// TIA Portal V20 export
FUNCTION_BLOCK "LER_StackMainCommand"   // FB95, LAD
// stored: Access Published, MemoryReserve 100, SetENOAutomatically false
   VAR_INPUT
      enable : Bool;
      reset : Bool;
      rollerCathodePos : Bool;
      rollerAnodePos : Bool;
      timeOffSet { ExternalAccessible := 'False'; ExternalVisible := 'False'; ExternalWritable := 'False'} : Time;
      motionStatus : Struct
         StopRequest : Bool := FALSE;
         Busy : Struct
            TotalBusy : Bool;
            CalculateBusy : Bool;
            SemiStepBusy : Bool;
            FullStepBusy : Bool;
            AutoBusy : Bool;
            CycleStopBusy : Bool;
            FastStopBusy : Bool;
            ResetBusy : Bool;
         END_STRUCT;
         Done : Struct
            TotalDone : Bool;
            CalculateDone : Bool;
            SemiStepDone : Bool;
            FullStepDone : Bool;
            AutoDone : Bool;
            CycleStopDone : Bool;
            FastStopDone : Bool;
            ResetDone : Bool;
         END_STRUCT;
         Error : Bool := FALSE;
         ErrorID : DWord := 16#0000_0000;
         NowCmd : DInt := 0;
         BeforeCmd : DInt := 0;
         NowStep : DInt := 160;
         BeforeStep : DInt := 180;
      END_STRUCT;
      unitStatus : "LAF_typeUnitStatus";
   END_VAR
   VAR_OUTPUT
      direction : Bool;
      motionCommands : Struct
         Calculate : Bool := FALSE;
         SemiStep : Bool := FALSE;
         FullStep : Bool := FALSE;
         Auto : Bool := FALSE;
         SepaClean : Bool;
         CycleStop : Bool := FALSE;
         FastStop : Bool;
         Reset : Bool := FALSE;
      END_STRUCT;
   END_VAR
   VAR_IN_OUT
      motionInterface : Struct
         Calculate : Bool;
         SemiStep : Bool;
         FullStep : Bool;
         AutoReady : Bool;
         AutoStart : Bool;
         StopMotion : Bool;
         StopForCalculate : Bool;
         Reset : Bool;
      END_STRUCT;
   END_VAR
   VAR
      statTonTime { ExternalAccessible := 'False'; ExternalVisible := 'False'; ExternalWritable := 'False'} : Array[0..999] of TON_TIME;
      statPulse { ExternalAccessible := 'False'; ExternalVisible := 'False'; ExternalWritable := 'False'} : Array[0..999] of Bool;
      statAction { ExternalAccessible := 'False'; ExternalVisible := 'False'; ExternalWritable := 'False'} : Array[0..999] of Bool;
      statStep { ExternalAccessible := 'False'; ExternalVisible := 'False'; ExternalWritable := 'False'} : DInt;
      statMotionStatus { ExternalAccessible := 'False'; ExternalVisible := 'False'; ExternalWritable := 'False'} : DInt;
   END_VAR
   VAR CONSTANT
      delayTime : Time := T#0ms;
   END_VAR
   VAR_TEMP   // added for the SCL form of the ladder/FBD networks
      _w1 : Bool;
      _w2 : Bool;
      _w3 : Bool;
      _w4 : Bool;
      _w5 : Bool;
      _w6 : Bool;
   END_VAR
BEGIN

REGION Network 1: ******************** Motion Operation ********************
END_REGION

REGION Network 2: STEP[0] : Motion Operation Condition
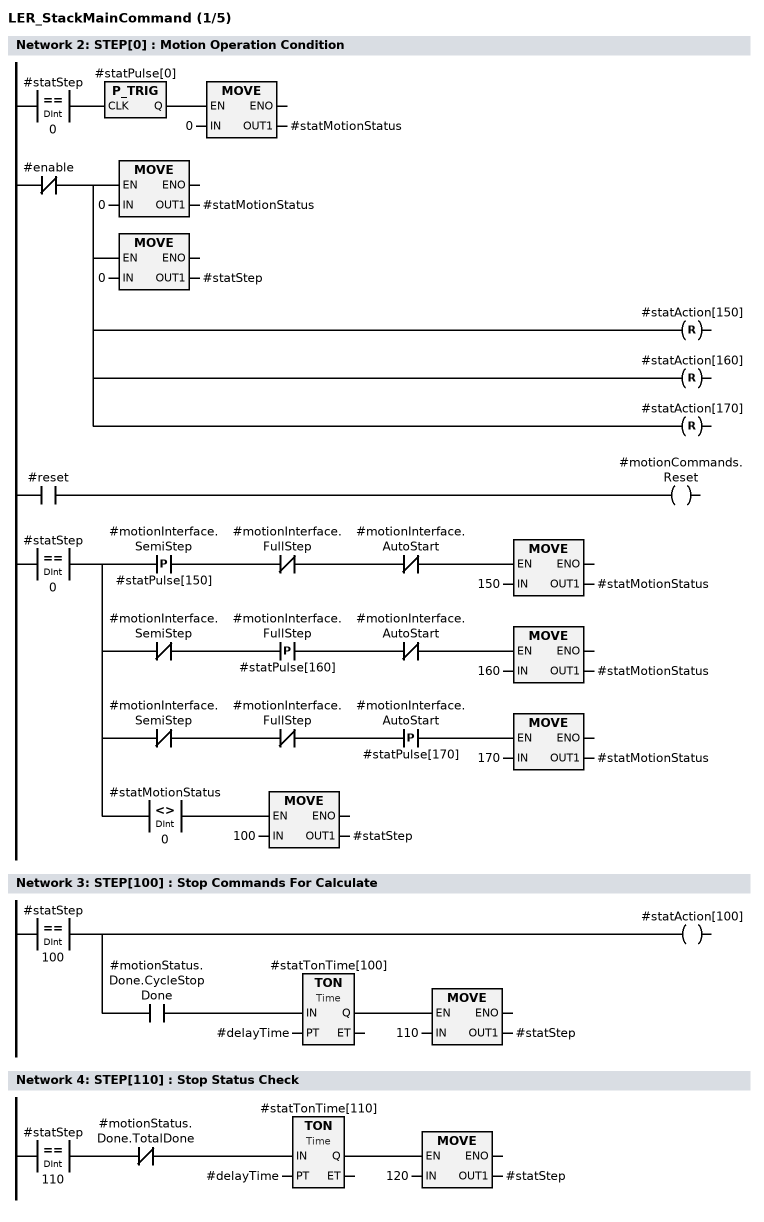
   RUNG wire#powerrail
      { S7_Templates := "SrcType := DInt" } EQ_Contact(in1 := #statStep, in2 := 0)
      P_Trig( #statPulse[0] )
      Move(in := 0, out1 => #statMotionStatus)
   END_RUNG
   RUNG wire#powerrail
      I_Contact( #enable )
      wire#w1
      Move(in := 0, out1 => #statMotionStatus)
   END_RUNG
   RUNG wire#w1
      Move(in := 0, out1 => #statStep)
   END_RUNG
   RUNG wire#w1
      R_Coil( #statAction[150] )
   END_RUNG
   RUNG wire#w1
      R_Coil( #statAction[160] )
   END_RUNG
   RUNG wire#w1
      R_Coil( #statAction[170] )
   END_RUNG
   RUNG wire#powerrail
      Contact( #reset )
      Coil( #motionCommands.Reset )
   END_RUNG
   RUNG wire#powerrail
      { S7_Templates := "SrcType := DInt" } EQ_Contact(in1 := #statStep, in2 := 0)
      wire#w2
      P_Contact(operand := #motionInterface.SemiStep, bit := #statPulse[150])
      I_Contact( #motionInterface.FullStep )
      I_Contact( #motionInterface.AutoStart )
      Move(in := 150, out1 => #statMotionStatus)
   END_RUNG
   RUNG wire#w2
      I_Contact( #motionInterface.SemiStep )
      P_Contact(operand := #motionInterface.FullStep, bit := #statPulse[160])
      I_Contact( #motionInterface.AutoStart )
      Move(in := 160, out1 => #statMotionStatus)
   END_RUNG
   RUNG wire#w2
      I_Contact( #motionInterface.SemiStep )
      I_Contact( #motionInterface.FullStep )
      P_Contact(operand := #motionInterface.AutoStart, bit := #statPulse[170])
      Move(in := 170, out1 => #statMotionStatus)
   END_RUNG
   RUNG wire#w2
      { S7_Templates := "SrcType := DInt" } NE_Contact(in1 := #statMotionStatus, in2 := 0)
      Move(in := 100, out1 => #statStep)
   END_RUNG
   // the same network as SCL:
   #_w1 := #statStep = 0;
   #_w2 := #_w1 AND NOT #statPulse[0];   // rising edge
   #statPulse[0] := #_w1;
   IF #_w2 THEN #statMotionStatus := 0; END_IF;
   IF NOT #enable THEN
       #statMotionStatus := 0;
       #statStep := 0;
       #statAction[150] := FALSE;
       #statAction[160] := FALSE;
       #statAction[170] := FALSE;
   END_IF;
   #motionCommands.Reset := #reset;
   #_w3 := #statStep = 0;
   #_w4 := #_w3 AND #motionInterface.SemiStep AND NOT #statPulse[150];   // rising edge of #motionInterface.SemiStep
   #statPulse[150] := #motionInterface.SemiStep;
   IF #_w4 AND NOT #motionInterface.FullStep AND NOT #motionInterface.AutoStart THEN
       #statMotionStatus := 150;
   END_IF;
   #_w5 := #_w3 AND NOT #motionInterface.SemiStep AND #motionInterface.FullStep AND NOT #statPulse[160];   // rising edge of #motionInterface.FullStep
   #statPulse[160] := #motionInterface.FullStep;
   IF #_w5 AND NOT #motionInterface.AutoStart THEN #statMotionStatus := 160; END_IF;
   #_w6 := #_w3 AND NOT #motionInterface.SemiStep AND NOT #motionInterface.FullStep AND #motionInterface.AutoStart AND NOT #statPulse[170];   // rising edge of #motionInterface.AutoStart
   #statPulse[170] := #motionInterface.AutoStart;
   IF #_w6 THEN #statMotionStatus := 170; END_IF;
   IF #_w3 AND (#statMotionStatus <> 0) THEN #statStep := 100; END_IF;
END_REGION

REGION Network 3: STEP[100] : Stop Commands For Calculate
   RUNG wire#powerrail
      { S7_Templates := "SrcType := DInt" } EQ_Contact(in1 := #statStep, in2 := 100)
      wire#w1
      Coil( #statAction[100] )
   END_RUNG
   RUNG wire#w1
      Contact( #motionStatus.Done.CycleStopDone )
      { S7_Templates := "time_type := Time" } #statTonTime[100].TON(pt := #delayTime, et =>)
      Move(in := 110, out1 => #statStep)
   END_RUNG
   // the same network as SCL:
   #statAction[100] := #statStep = 100;
   #statTonTime[100].TON(IN := (#statStep = 100) AND #motionStatus.Done.CycleStopDone, PT := #delayTime);
   IF #statTonTime[100].Q THEN #statStep := 110; END_IF;
END_REGION

REGION Network 4: STEP[110] : Stop Status Check
   RUNG wire#powerrail
      { S7_Templates := "SrcType := DInt" } EQ_Contact(in1 := #statStep, in2 := 110)
      I_Contact( #motionStatus.Done.TotalDone )
      { S7_Templates := "time_type := Time" } #statTonTime[110].TON(pt := #delayTime, et =>)
      Move(in := 120, out1 => #statStep)
   END_RUNG
   // the same network as SCL:
   #statTonTime[110].TON(IN := (#statStep = 110) AND NOT #motionStatus.Done.TotalDone, PT := #delayTime);
   IF #statTonTime[110].Q THEN #statStep := 120; END_IF;
END_REGION

REGION Network 5: STEP[120] : Parameter Direction Select
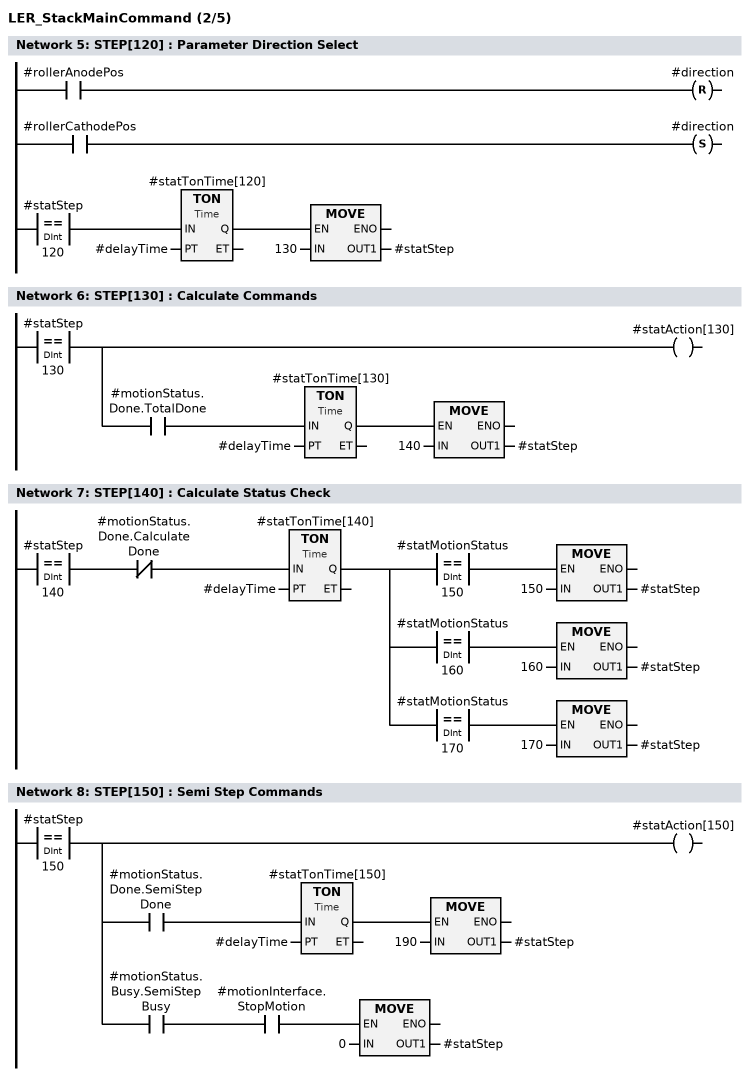
   RUNG wire#powerrail
      Contact( #rollerAnodePos )
      R_Coil( #direction )
   END_RUNG
   RUNG wire#powerrail
      Contact( #rollerCathodePos )
      S_Coil( #direction )
   END_RUNG
   RUNG wire#powerrail
      { S7_Templates := "SrcType := DInt" } EQ_Contact(in1 := #statStep, in2 := 120)
      { S7_Templates := "time_type := Time" } #statTonTime[120].TON(pt := #delayTime, et =>)
      Move(in := 130, out1 => #statStep)
   END_RUNG
   // the same network as SCL:
   IF #rollerAnodePos THEN #direction := FALSE; END_IF;
   IF #rollerCathodePos THEN #direction := TRUE; END_IF;
   #statTonTime[120].TON(IN := #statStep = 120, PT := #delayTime);
   IF #statTonTime[120].Q THEN #statStep := 130; END_IF;
END_REGION

REGION Network 6: STEP[130] : Calculate Commands
   RUNG wire#powerrail
      { S7_Templates := "SrcType := DInt" } EQ_Contact(in1 := #statStep, in2 := 130)
      wire#w1
      Coil( #statAction[130] )
   END_RUNG
   RUNG wire#w1
      Contact( #motionStatus.Done.TotalDone )
      { S7_Templates := "time_type := Time" } #statTonTime[130].TON(pt := #delayTime, et =>)
      Move(in := 140, out1 => #statStep)
   END_RUNG
   // the same network as SCL:
   #statAction[130] := #statStep = 130;
   #statTonTime[130].TON(IN := (#statStep = 130) AND #motionStatus.Done.TotalDone, PT := #delayTime);
   IF #statTonTime[130].Q THEN #statStep := 140; END_IF;
END_REGION

REGION Network 7: STEP[140] : Calculate Status Check
   RUNG wire#powerrail
      { S7_Templates := "SrcType := DInt" } EQ_Contact(in1 := #statStep, in2 := 140)
      I_Contact( #motionStatus.Done.CalculateDone )
      { S7_Templates := "time_type := Time" } #statTonTime[140].TON(pt := #delayTime, et =>)
      wire#w1
      { S7_Templates := "SrcType := DInt" } EQ_Contact(in1 := #statMotionStatus, in2 := 150)
      Move(in := 150, out1 => #statStep)
   END_RUNG
   RUNG wire#w1
      { S7_Templates := "SrcType := DInt" } EQ_Contact(in1 := #statMotionStatus, in2 := 160)
      Move(in := 160, out1 => #statStep)
   END_RUNG
   RUNG wire#w1
      { S7_Templates := "SrcType := DInt" } EQ_Contact(in1 := #statMotionStatus, in2 := 170)
      Move(in := 170, out1 => #statStep)
   END_RUNG
   // the same network as SCL:
   #statTonTime[140].TON(IN := (#statStep = 140) AND NOT #motionStatus.Done.CalculateDone, PT := #delayTime);
   IF #statTonTime[140].Q AND (#statMotionStatus = 150) THEN #statStep := 150; END_IF;
   IF #statTonTime[140].Q AND (#statMotionStatus = 160) THEN #statStep := 160; END_IF;
   IF #statTonTime[140].Q AND (#statMotionStatus = 170) THEN #statStep := 170; END_IF;
END_REGION

REGION Network 8: STEP[150] : Semi Step Commands
   RUNG wire#powerrail
      { S7_Templates := "SrcType := DInt" } EQ_Contact(in1 := #statStep, in2 := 150)
      wire#w1
      Coil( #statAction[150] )
   END_RUNG
   RUNG wire#w1
      Contact( #motionStatus.Done.SemiStepDone )
      { S7_Templates := "time_type := Time" } #statTonTime[150].TON(pt := #delayTime, et =>)
      Move(in := 190, out1 => #statStep)
   END_RUNG
   RUNG wire#w1
      Contact( #motionStatus.Busy.SemiStepBusy )
      Contact( #motionInterface.StopMotion )
      Move(in := 0, out1 => #statStep)
   END_RUNG
   // the same network as SCL:
   #statAction[150] := #statStep = 150;
   #statTonTime[150].TON(IN := (#statStep = 150) AND #motionStatus.Done.SemiStepDone, PT := #delayTime);
   #_w1 := #statStep = 150;
   IF #statTonTime[150].Q THEN #statStep := 190; END_IF;
   IF #_w1 AND #motionStatus.Busy.SemiStepBusy AND #motionInterface.StopMotion THEN #statStep := 0; END_IF;
END_REGION

REGION Network 9: STEP[160] : Full Step Commands
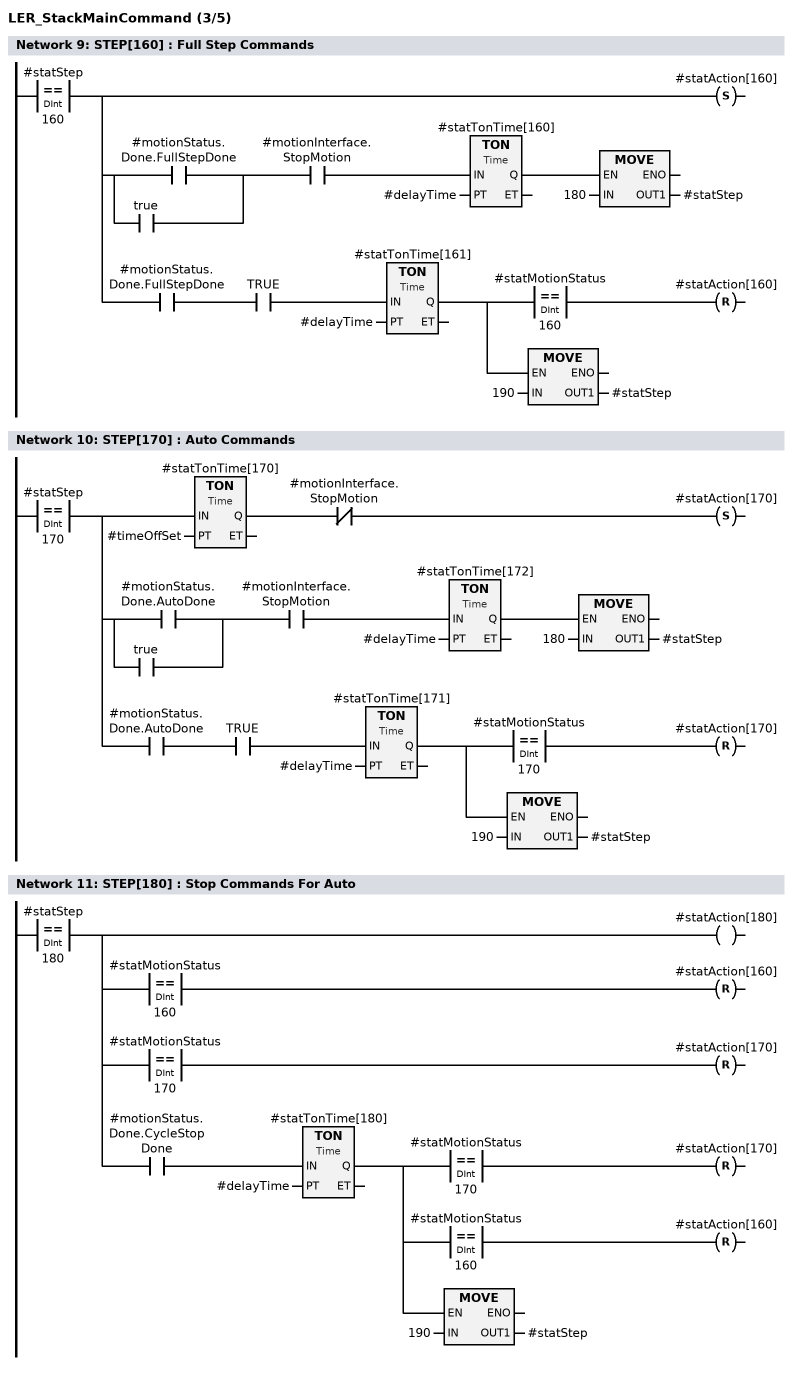
   RUNG wire#powerrail
      { S7_Templates := "SrcType := DInt" } EQ_Contact(in1 := #statStep, in2 := 160)
      wire#w1
      S_Coil( #statAction[160] )
   END_RUNG
   RUNG wire#w1
      Contact( #motionStatus.Done.FullStepDone )
      wire#w2
      Contact( #motionInterface.StopMotion )
      { S7_Templates := "time_type := Time" } #statTonTime[160].TON(pt := #delayTime, et =>)
      Move(in := 180, out1 => #statStep)
   END_RUNG
   RUNG wire#w1
      Contact( true )
   END_RUNG wire#w2
   RUNG wire#w1
      Contact( #motionStatus.Done.FullStepDone )
      Contact( TRUE )
      { S7_Templates := "time_type := Time" } #statTonTime[161].TON(pt := #delayTime, et =>)
      wire#w3
      { S7_Templates := "SrcType := DInt" } EQ_Contact(in1 := #statMotionStatus, in2 := 160)
      R_Coil( #statAction[160] )
   END_RUNG
   RUNG wire#w3
      Move(in := 190, out1 => #statStep)
   END_RUNG
   // the same network as SCL:
   #_w1 := #statStep = 160;
   IF #_w1 THEN #statAction[160] := TRUE; END_IF;
   #statTonTime[160].TON(IN := #_w1 AND (#motionStatus.Done.FullStepDone OR true) AND #motionInterface.StopMotion,
                         PT := #delayTime);
   IF #statTonTime[160].Q THEN #statStep := 180; END_IF;
   #statTonTime[161].TON(IN := #_w1 AND #motionStatus.Done.FullStepDone AND TRUE, PT := #delayTime);
   IF #statTonTime[161].Q AND (#statMotionStatus = 160) THEN #statAction[160] := FALSE; END_IF;
   IF #statTonTime[161].Q THEN #statStep := 190; END_IF;
END_REGION

REGION Network 10: STEP[170] : Auto Commands
   RUNG wire#powerrail
      { S7_Templates := "SrcType := DInt" } EQ_Contact(in1 := #statStep, in2 := 170)
      wire#w1
      { S7_Templates := "time_type := Time" } #statTonTime[170].TON(pt := #timeOffSet, et =>)
      I_Contact( #motionInterface.StopMotion )
      S_Coil( #statAction[170] )
   END_RUNG
   RUNG wire#w1
      Contact( #motionStatus.Done.AutoDone )
      wire#w2
      Contact( #motionInterface.StopMotion )
      { S7_Templates := "time_type := Time" } #statTonTime[172].TON(pt := #delayTime, et =>)
      Move(in := 180, out1 => #statStep)
   END_RUNG
   RUNG wire#w1
      Contact( true )
   END_RUNG wire#w2
   RUNG wire#w1
      Contact( #motionStatus.Done.AutoDone )
      Contact( TRUE )
      { S7_Templates := "time_type := Time" } #statTonTime[171].TON(pt := #delayTime, et =>)
      wire#w3
      { S7_Templates := "SrcType := DInt" } EQ_Contact(in1 := #statMotionStatus, in2 := 170)
      R_Coil( #statAction[170] )
   END_RUNG
   RUNG wire#w3
      Move(in := 190, out1 => #statStep)
   END_RUNG
   // the same network as SCL:
   #_w1 := #statStep = 170;
   #statTonTime[170].TON(IN := #_w1, PT := #timeOffSet);
   IF #statTonTime[170].Q AND NOT #motionInterface.StopMotion THEN #statAction[170] := TRUE; END_IF;
   #statTonTime[172].TON(IN := #_w1 AND (#motionStatus.Done.AutoDone OR true) AND #motionInterface.StopMotion,
                         PT := #delayTime);
   IF #statTonTime[172].Q THEN #statStep := 180; END_IF;
   #statTonTime[171].TON(IN := #_w1 AND #motionStatus.Done.AutoDone AND TRUE, PT := #delayTime);
   IF #statTonTime[171].Q AND (#statMotionStatus = 170) THEN #statAction[170] := FALSE; END_IF;
   IF #statTonTime[171].Q THEN #statStep := 190; END_IF;
END_REGION

REGION Network 11: STEP[180] : Stop Commands For Auto
   RUNG wire#powerrail
      { S7_Templates := "SrcType := DInt" } EQ_Contact(in1 := #statStep, in2 := 180)
      wire#w1
      Coil( #statAction[180] )
   END_RUNG
   RUNG wire#w1
      { S7_Templates := "SrcType := DInt" } EQ_Contact(in1 := #statMotionStatus, in2 := 160)
      R_Coil( #statAction[160] )
   END_RUNG
   RUNG wire#w1
      { S7_Templates := "SrcType := DInt" } EQ_Contact(in1 := #statMotionStatus, in2 := 170)
      R_Coil( #statAction[170] )
   END_RUNG
   RUNG wire#w1
      Contact( #motionStatus.Done.CycleStopDone )
      { S7_Templates := "time_type := Time" } #statTonTime[180].TON(pt := #delayTime, et =>)
      wire#w2
      { S7_Templates := "SrcType := DInt" } EQ_Contact(in1 := #statMotionStatus, in2 := 170)
      R_Coil( #statAction[170] )
   END_RUNG
   RUNG wire#w2
      { S7_Templates := "SrcType := DInt" } EQ_Contact(in1 := #statMotionStatus, in2 := 160)
      R_Coil( #statAction[160] )
   END_RUNG
   RUNG wire#w2
      Move(in := 190, out1 => #statStep)
   END_RUNG
   // the same network as SCL:
   #statAction[180] := #statStep = 180;
   IF (#statStep = 180) AND (#statMotionStatus = 160) THEN #statAction[160] := FALSE; END_IF;
   IF (#statStep = 180) AND (#statMotionStatus = 170) THEN #statAction[170] := FALSE; END_IF;
   #statTonTime[180].TON(IN := (#statStep = 180) AND #motionStatus.Done.CycleStopDone, PT := #delayTime);
   IF #statTonTime[180].Q AND (#statMotionStatus = 170) THEN #statAction[170] := FALSE; END_IF;
   IF #statTonTime[180].Q AND (#statMotionStatus = 160) THEN #statAction[160] := FALSE; END_IF;
   IF #statTonTime[180].Q THEN #statStep := 190; END_IF;
END_REGION

REGION Network 12: STEP[190] : Motion Operation Complete
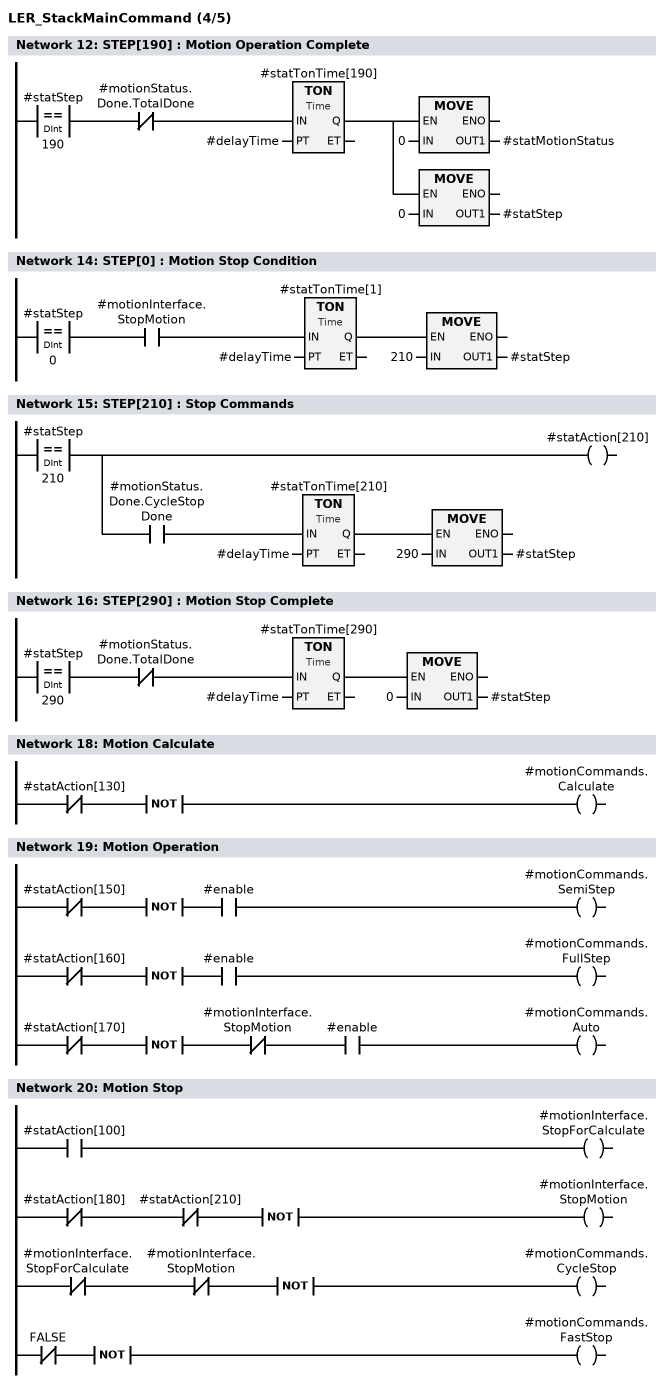
   RUNG wire#powerrail
      { S7_Templates := "SrcType := DInt" } EQ_Contact(in1 := #statStep, in2 := 190)
      I_Contact( #motionStatus.Done.TotalDone )
      { S7_Templates := "time_type := Time" } #statTonTime[190].TON(pt := #delayTime, et =>)
      wire#w1
      Move(in := 0, out1 => #statMotionStatus)
   END_RUNG
   RUNG wire#w1
      Move(in := 0, out1 => #statStep)
   END_RUNG
   // the same network as SCL:
   #statTonTime[190].TON(IN := (#statStep = 190) AND NOT #motionStatus.Done.TotalDone, PT := #delayTime);
   IF #statTonTime[190].Q THEN
       #statMotionStatus := 0;
       #statStep := 0;
   END_IF;
END_REGION

REGION Network 13: ******************** Motion Stop ********************
END_REGION

REGION Network 14: STEP[0] : Motion Stop Condition
   RUNG wire#powerrail
      { S7_Templates := "SrcType := DInt" } EQ_Contact(in1 := #statStep, in2 := 0)
      Contact( #motionInterface.StopMotion )
      { S7_Templates := "time_type := Time" } #statTonTime[1].TON(pt := #delayTime, et =>)
      Move(in := 210, out1 => #statStep)
   END_RUNG
   // the same network as SCL:
   #statTonTime[1].TON(IN := (#statStep = 0) AND #motionInterface.StopMotion, PT := #delayTime);
   IF #statTonTime[1].Q THEN #statStep := 210; END_IF;
END_REGION

REGION Network 15: STEP[210] : Stop Commands
   RUNG wire#powerrail
      { S7_Templates := "SrcType := DInt" } EQ_Contact(in1 := #statStep, in2 := 210)
      wire#w1
      Coil( #statAction[210] )
   END_RUNG
   RUNG wire#w1
      Contact( #motionStatus.Done.CycleStopDone )
      { S7_Templates := "time_type := Time" } #statTonTime[210].TON(pt := #delayTime, et =>)
      Move(in := 290, out1 => #statStep)
   END_RUNG
   // the same network as SCL:
   #statAction[210] := #statStep = 210;
   #statTonTime[210].TON(IN := (#statStep = 210) AND #motionStatus.Done.CycleStopDone, PT := #delayTime);
   IF #statTonTime[210].Q THEN #statStep := 290; END_IF;
END_REGION

REGION Network 16: STEP[290] : Motion Stop Complete
   RUNG wire#powerrail
      { S7_Templates := "SrcType := DInt" } EQ_Contact(in1 := #statStep, in2 := 290)
      I_Contact( #motionStatus.Done.TotalDone )
      { S7_Templates := "time_type := Time" } #statTonTime[290].TON(pt := #delayTime, et =>)
      Move(in := 0, out1 => #statStep)
   END_RUNG
   // the same network as SCL:
   #statTonTime[290].TON(IN := (#statStep = 290) AND NOT #motionStatus.Done.TotalDone, PT := #delayTime);
   IF #statTonTime[290].Q THEN #statStep := 0; END_IF;
END_REGION

REGION Network 17: ******************** Motion Commands ********************
END_REGION

REGION Network 18: Motion Calculate
   RUNG wire#powerrail
      I_Contact( #statAction[130] )
      Not()
      Coil( #motionCommands.Calculate )
   END_RUNG
   // the same network as SCL:
   #motionCommands.Calculate := NOT (NOT #statAction[130]);
END_REGION

REGION Network 19: Motion Operation
   RUNG wire#powerrail
      I_Contact( #statAction[150] )
      Not()
      Contact( #enable )
      Coil( #motionCommands.SemiStep )
   END_RUNG
   RUNG wire#powerrail
      I_Contact( #statAction[160] )
      Not()
      Contact( #enable )
      Coil( #motionCommands.FullStep )
   END_RUNG
   RUNG wire#powerrail
      I_Contact( #statAction[170] )
      Not()
      I_Contact( #motionInterface.StopMotion )
      Contact( #enable )
      Coil( #motionCommands.Auto )
   END_RUNG
   // the same network as SCL:
   #motionCommands.SemiStep := NOT (NOT #statAction[150]) AND #enable;
   #motionCommands.FullStep := NOT (NOT #statAction[160]) AND #enable;
   #motionCommands.Auto := NOT (NOT #statAction[170]) AND NOT #motionInterface.StopMotion AND #enable;
END_REGION

REGION Network 20: Motion Stop
   RUNG wire#powerrail
      Contact( #statAction[100] )
      Coil( #motionInterface.StopForCalculate )
   END_RUNG
   RUNG wire#powerrail
      I_Contact( #statAction[180] )
      I_Contact( #statAction[210] )
      Not()
      Coil( #motionInterface.StopMotion )
   END_RUNG
   RUNG wire#powerrail
      I_Contact( #motionInterface.StopForCalculate )
      I_Contact( #motionInterface.StopMotion )
      Not()
      Coil( #motionCommands.CycleStop )
   END_RUNG
   RUNG wire#powerrail
      I_Contact( FALSE )
      Not()
      Coil( #motionCommands.FastStop )
   END_RUNG
   // the same network as SCL:
   #motionInterface.StopForCalculate := #statAction[100];
   #motionInterface.StopMotion := NOT (NOT #statAction[180] AND NOT #statAction[210]);
   #motionCommands.CycleStop := NOT (NOT #motionInterface.StopForCalculate AND NOT #motionInterface.StopMotion);
   #motionCommands.FastStop := NOT (NOT FALSE);
END_REGION

REGION Network 21: Motion Reset
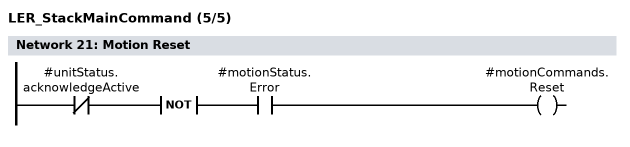
   RUNG wire#powerrail
      I_Contact( #unitStatus.acknowledgeActive )
      Not()
      Contact( #motionStatus.Error )
      Coil( #motionCommands.Reset )
   END_RUNG
   // the same network as SCL:
   #motionCommands.Reset := NOT (NOT #unitStatus.acknowledgeActive) AND #motionStatus.Error;
END_REGION

REGION Network 22: ******************** Function Commands ********************
END_REGION

REGION Network 23: Function Reset
END_REGION
END_FUNCTION_BLOCK
